// TIA Portal V17 export
// export: Created 2025-02-20T16:06:01.3767978Z, ExportSetting WithDefaults, DisplayName Totally Integrated Automation Portal, DisplayVersion V17 Update 6, DisplayName TIA Portal Openness, DisplayVersion V17 Update 6, DisplayName TIA Portal Version Control Interface, DisplayVersion V17, DisplayName STEP 7 Professional, DisplayVersion V17 Update 6, DisplayName STEP 7 Safety, DisplayVersion V17 Update 6, DisplayName WinCC Advanced, DisplayVersion V17 Update 6
FUNCTION "ARRANQUE DE MOTOR" : Void   // FC1, LAD
{ S7_Optimized_Access := 'TRUE' }
VERSION : 0.1
// stored: AutoNumber true, IsIECCheckEnabled false, SetENOAutomatically false, UDAEnableTagReadback false
BEGIN

REGION Network 1
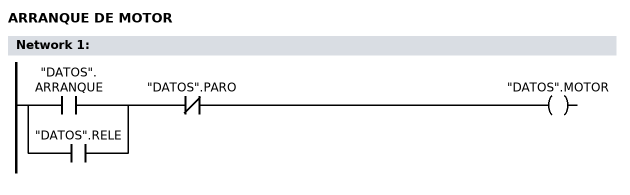
   RUNG wire#powerrail
      Contact( "DATOS".ARRANQUE )
      wire#w1
      I_Contact( "DATOS".PARO )
      Coil( "DATOS".MOTOR )
   END_RUNG
   RUNG wire#powerrail
      Contact( "DATOS".RELE )
   END_RUNG wire#w1
   // the same network as SCL:
   "DATOS".MOTOR := ("DATOS".ARRANQUE OR "DATOS".RELE) AND NOT "DATOS".PARO;
END_REGION
END_FUNCTION
